// TIA Portal V17 export
// export: Created 2022-03-12T16:05:30.8407121Z, ExportSetting WithDefaults, DisplayName Totally Integrated Automation Portal, DisplayVersion V17, DisplayName TIA Portal Openness, DisplayVersion V17, DisplayName TIA Portal Version Control Interface, DisplayVersion V17, DisplayName STEP 7 Professional, DisplayVersion V17, DisplayName STEP 7 Safety, DisplayVersion V17, DisplayName WinCC Advanced / Unified PC, DisplayVersion V17
DATA_BLOCK "PackTags"   // DB31614
TITLE = CPG_PackTags
{ S7_Optimized_Access := 'TRUE' }
AUTHOR : tech.team.motioncontrol@siemens.com
FAMILY : CPG
VERSION : 1.0
// Support: tech.team.motioncontrol@siemens.com
// Fax: +49 (0) 9131/98-1297
// stored: AutoNumber true, DBAccessibleFromOPCUA true, DBAccessibleFromWebserver true, IsOnlyStoredInLoadMemory false, IsRetainMemResEnabled false, IsWriteProtectedInAS false, MemoryReserve 0
   VAR
      Command : Struct   // PackTags "Command" tag area. Data is scalable for needs.
         UnitMode : DInt;   // Unit Mode Target (1=Production,2=Maintenance,3=Manual,4=UserMode1,...,31=UserMode28)
         UnitModeChangeRequest : Bool;   // 1=Request Unit Mode Change to commanded value (UnitMode)
         MachSpeed : Real := 0.0;   // Setpoint of Machine Speed in Primary Packages per Minute
         MaterialInterlock : DWord;   // Materials Interlock Command (1=Ready or Not low, 0=Not ready or Low)
         CntrlCmd : DInt;   // State Control Command to drive a state change (1=Reset,2=Start,3=Stop,4=Hold,5=Unhold,6=Suspend,7=Unsuspend,8=Abort,9=Clear)
         CmdChangeRequest : Bool;   // 1=Request Machine State Change to commanded value (CntrlCmd)
         Parameter { S7_SetPoint := 'True'} : Array[0.."CPG_NO_OF_COMMAND_PARAMETERS_UPPER_LIM"] of "CPG_typeParameter(Real)";   // Parameter Structure Array from SCADA / MES
      END_STRUCT;
      Status { ExternalWritable := 'False'} : Struct   // PackTags "Status" tag area. Data is scalable for needs.
         UnitModeCurrent { ExternalWritable := 'False'} : DInt := 3;   // Current Unit Mode (1=Production,2=Maintenance,3=Manual,4=UserMode1,...,31=UserMode28)
         UnitModeCurrentName { ExternalWritable := 'False'} : String[18] := 'Manual';   // Current Unit Mode Name (NOT ISA-TR88 - OPTIONAL)
         UnitModeRequested { ExternalWritable := 'False'} : Bool;   // 1=Ack. that a unit mode change has been requested
         UnitModeChangeInProcess { ExternalWritable := 'False'} : Bool;   // 1=Requested Unit Mode Change In Progress
         StateCurrent { ExternalWritable := 'False'} : DInt := 2;   // Current Machine State (1=Clearing,2=Stopped,3=Starting,4=Idle,5=Suspended,6=Execute,7=Stopping,8=Aborting,9=Aborted,10=Holding,11=Held,12=Unholding,13=Suspending,14=Unsuspending,15=Resetting,16=Completing,17=Complete)
         StateCurrentName { ExternalWritable := 'False'} : String[16] := 'Stopped';   // Current Machine State name (NOT ISA-TR88 - OPTIONAL)
         StateRequested { ExternalWritable := 'False'} : DInt;   // Target Machine State
         StateChangeInProcess { ExternalWritable := 'False'} : Bool;   // 1=Requested State Change in Progress
         MachSpeed { ExternalWritable := 'False'} : Real := 0.0;   // Setpoint of Machine Speed in Primary Packages per Minute
         CurMachSpeed { ExternalWritable := 'False'} : Real := 0.0;   // Actual Value of Machine Speed in Primary Packages per Minute
         MaterialInterlock { ExternalWritable := 'False'} : DWord;   // Materials Interlock Status (1=Ready or Not low, 0=Not ready or Low)
         EquipmentInterlock { ExternalWritable := 'False'} : Struct   // Machine upstream and downstream status
            Blocked { ExternalWritable := 'False'} : Bool;   // 1=The downstream system is not able to accept products, 0=all OK
            Starved { ExternalWritable := 'False'} : Bool;   // 1=The upstream system is not able to supply products, 0=all OK
         END_STRUCT;
         Parameter { ExternalWritable := 'False'; S7_SetPoint := 'True'} : Array[0.."CPG_NO_OF_STATUS_PARAMETERS_UPPER_LIM"] of "CPG_typeParameter(Real)";   // Parameter Structure Array for HMI / SCADA / MES
      END_STRUCT;
   END_VAR
   VAR RETAIN
      Admin { ExternalWritable := 'False'} : Struct   // PackTags "Administration" tag area. Data is scalable for needs.
         Parameter { ExternalWritable := 'False'; S7_SetPoint := 'True'} : Array[0.."CPG_NO_OF_ADMIN_PARAMETERS_UPPER_LIM"] of "CPG_typeParameter(Real)";   // Parameter Structure Array for HMI / SCADA / MES
         Alarm { ExternalWritable := 'False'; S7_SetPoint := 'True'} : Array[0.."CPG_NO_OF_ADMIN_EVENTS_UPPER_LIM"] of "CPG_typeEvent";   // Alarm summary of Active Events
         AlarmExtent { ExternalWritable := 'False'} : DInt;   // Number of active alarms
         AlarmHistory { ExternalWritable := 'False'; S7_SetPoint := 'True'} : Array[0.."CPG_NO_OF_ADMIN_EVENTS_HISTORY_UPPER_LIM"] of "CPG_typeEvent";   // Alarm History
         AlarmHistoryExtent { ExternalWritable := 'False'} : DInt;   // Number of alarms in alarm history
         StopReason { ExternalWritable := 'False'; S7_SetPoint := 'True'} : "CPG_typeEvent";   // First Fault Alarm Code
         Warning { ExternalWritable := 'False'; S7_SetPoint := 'True'} : Array[0.."CPG_NO_OF_ADMIN_EVENTS_UPPER_LIM"] of "CPG_typeEvent";   // Active Machine Warnings
         WarningExtent { ExternalWritable := 'False'} : DInt;   // Number of Active Machine Warnings
         ModeCurrentTime { ExternalWritable := 'False'} : Array[0.."LPMLV30_MODES_UPPER_LIM"] of DInt;   // Time spent in the last mode [seconds] (reset each time new mode is entered)
         ModeCumulativeTime { ExternalWritable := 'False'} : Array[0.."LPMLV30_MODES_UPPER_LIM"] of DInt;   // Cumulative Time for all Modes [seconds]
         StateCurrentTime { ExternalWritable := 'False'} : Array[0.."LPMLV30_MODES_UPPER_LIM", 0.."LPMLV30_STATES_UPPER_LIM"] of DInt;   // Time spent in the last state [seconds] (reset each time new state is entered)
         StateCumulativeTime { ExternalWritable := 'False'} : Array[0.."LPMLV30_MODES_UPPER_LIM", 0.."LPMLV30_STATES_UPPER_LIM"] of DInt;   // Cumulative Time for all States [seconds]
         ProdConsumedCount { ExternalWritable := 'False'; S7_SetPoint := 'True'} : Array[0.."CPG_NO_OF_PROD_CONSUMED_COUNT_UPPER_LIM"] of "CPG_typeProdCount(DINT)";   // Total Number of Products consumed- good or bad
         ProdProcessedCount { ExternalWritable := 'False'; S7_SetPoint := 'True'} : Array[0.."CPG_NO_OF_PROD_PROCESSED_COUNT_UPPER_LIM"] of "CPG_typeProdCount(DINT)";   // Total Number of Products processed - good or bad
         ProdDefectiveCount { ExternalWritable := 'False'; S7_SetPoint := 'True'} : Array[0.."CPG_NO_OF_PROD_DEFECTIVE_COUNT_UPPER_LIM"] of "CPG_typeProdCount(DINT)";   // Total Number of Defective (bad) Products processed
         AccTimeSinceLastReset { ExternalWritable := 'False'} : DInt := L#0;   // Accumulated Time Since Last Reset of all mode and state times and counts
         MachDesignSpeed { ExternalWritable := 'False'} : Real := 0.0;   // Machine Design Speed of the Current Product Configuration
         StatesDisabled { ExternalWritable := 'False'} : DInt;   // States 1 to 17 of the PackML State Model can be disabled by turning on the corresponding bit in the DINT
         PLCDateTime { ExternalWritable := 'False'} : Array[0..6] of DInt;   // Current Date and Time of PLC
         PLCDateTimeDTL { ExternalWritable := 'False'} : DTL;   // Current Date and LTime (DTL) of PLC (date and time-of-day information in nanoseconds since 01/01/1970 0:0)
      END_STRUCT;
   END_VAR
BEGIN
   Admin.ProdConsumedCount[0]."Name" := 'Consumed #1';
   Admin.ProdConsumedCount[0].Unit := 'count';
   Admin.ProdProcessedCount[0]."Name" := 'Processed #1';
   Admin.ProdProcessedCount[0].Unit := 'count';
   Admin.ProdDefectiveCount[0]."Name" := 'Defective #1';
   Admin.ProdDefectiveCount[0].Unit := 'count';
END_DATA_BLOCK
